FUNCTION_BLOCK Basic (* Basic Function Block Type *)
  (* Standard: 61499-2 *)
  (* Version 0.3, 2009-09-15, JHC, Holobloc Inc, Changed transition priorities. *)
  (* Version 0.2, 2003-12-04, JHC, Rockwell Automation, Renamed for better indexing. *)
  (* Version 0.1, 2002-11-05, JHC, Rockwell Automation, Corrected missing ST element in Algorithm REQ. *)
  (* Version 0.0, 2000-05-30, JHC, Rockwell Automation *)
  (* Compiler header: package fb.rt.template; *)
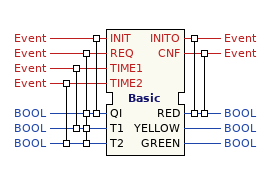
  EVENT_INPUT
    INIT WITH QI; (* Initialization Request *)
    REQ WITH QI, T1, T2; (* Normal Execution Request *)
    TIME1 WITH T1;
    TIME2 WITH T2;
  END_EVENT
  EVENT_OUTPUT
    INITO WITH RED; (* Initialization Confirm *)
    CNF WITH RED; (* Execution Confirmation *)
  END_EVENT
  VAR_INPUT
    QI : BOOL; (* Input event qualifier *)
    T1 : BOOL;
    T2 : BOOL;
  END_VAR
  VAR_OUTPUT
    RED : BOOL; (* Output event qualifier *)
    YELLOW : BOOL;
    GREEN : BOOL;
  END_VAR
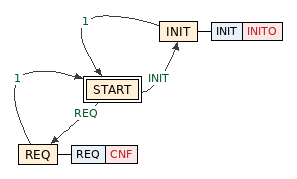
  EC_STATES
    START; (* Initial State *)
    INIT : INIT -> INITO; (* Initialization *)
    REQ : REQ -> CNF; (* Normal execution *)
  END_STATES
  EC_TRANSITIONS
    INIT TO START := 1;
    START TO REQ := REQ;
    START TO INIT := INIT;
    REQ TO START := 1;
  END_TRANSITIONS
  ALGORITHM INIT IN ST: (* Initialization algorithm *)
IF Q1 THEN
	GREEN:=FALSE;
	Yellow:=FALSE;
	Red:=FALSE;
END_IF;
  END_ALGORITHM
  ALGORITHM REQ IN ST: (* Normally executed algorithm *)
IF QI THEN
	GREEN:=FALSE;
	YELLOW:=TRUE;
END_IF;
  END_ALGORITHM
  ALGORITHM TIME1 IN ST:
IF T1 THEN
	GREEN:=FALSE;
	YELLOW:=TRUE;
END_IF;
  END_ALGORITHM
  ALGORITHM TIME2 IN ST:
IF T2 THEN
	YELLOW:=FALSE;
	RED:=TRUE;
END_IF;
  END_ALGORITHM
END_FUNCTION_BLOCK
